	23:
		bRunSteamBypass													:= P_U01.SP_steam_bypass_immediately_after_warm_up;
		IF bAdsorptionActive AND NOT bRunSteamBypass THEN 																	// 14
			i2Step														:= 30;
		ELSIF bAdsorptionActive AND bRunSteamBypass AND NOT P_U01.SP_adsorb_during_steam_bypass THEN
			i2Step														:= 40;												// 15
		ELSE
			i2Step														:= 90;												// 13 & 16
		END_IF
	
		
//**** Adsorption 1		
	30:
		IF tonAdsorptionTimer.Q THEN																						// 14.a
			bAdsorptionTimer											:= FALSE;
			gsCycleStage												:= 'warm_up.boiler_heating.turn_off_fans';			// 14.b
			P_M01.rs1.fan_setpoint										:= 0;												// 14.c
			rTime														:= _FAN_RS_DELAY_TIME;
			i2Step														:= i2Step + 1;
		END_IF

	31:
		bTimer															:= TRUE;
		IF tonTimer.Q THEN
			bTimer														:= FALSE;
			gsCycleStage												:= 'warm_up.boiler_heating.closing_doors';			// 14.d
			P_M01.rs1.close_doors										:= TRUE;											// 14.e
			rTime														:= P_M01.SP_doorsopenclose_timedelay * _MINUTES;										// 14.e.i
			i2Step														:= i2Step + 1;
		END_IF		

	32:
		bTimer															:= TRUE;
		bPass1															:= (P_M01.bRS01 AND P_M01.rs1.inlet_doors_closed AND P_M01.rs1.outlet_doors_closed) OR NOT P_M01.bRS01;	// 14.e.ii
		IF bPass1 THEN
			bTimer														:= FALSE;
			i2Step														:= i2Step + 1;
		ELSIF tonTimer.Q THEN																								// 14.e.i
			bTimer														:= FALSE;
			bRunSteamBypass												:= FALSE;
			sRS															:= _RS01;
			P_Alarms.M_Add_Alarm(F_Concat3(_U01, sRS, gsCycleStage), gsReactorDoorClosingError, gsSystemCannotRun);
			i2Step														:= i2Step + 1;
		END_IF
		
	33:
		//P_M01_RS01.co2_sensors_on										:= FALSE;											// 14.f
		bAdsorptionActive												:= FALSE;											// 14.g
		i2Step															:= 90;

	
//**** Adsorption 2	
	40:
		IF tonAdsorptionTimer.Q THEN																						// 15.a
			bAdsorptionTimer											:= FALSE;
			P_M01.rs1.fan_setpoint										:= 0;												// 15.b
			rTime														:= _FAN_RS_DELAY_TIME;
			i2Step														:= i2Step + 1;
		END_IF

	41:
		bTimer															:= TRUE;
		IF tonTimer.Q THEN
			bTimer														:= FALSE;											// 15.c
			//P_M01_RS01.co2_sensors_on									:= FALSE;
			bAdsorptionActive											:= FALSE;											// 15.d
			i2Step														:= i2Step + 1;
		END_IF
		
	42:
		P_M01.rs1.close_doors											:= TRUE;											// 15.g
		rTime															:= P_M01.SP_doorsopenclose_timedelay * _MINUTES;										// 15.g.i
		i2Step															:= i2Step + 1;

	43:
		bTimer															:= TRUE;
		bPass1															:= (P_M01.bRS01 AND P_M01.rs1.inlet_doors_closed AND P_M01.rs1.outlet_doors_closed) OR NOT P_M01.bRS01;		// 15.g.ii
		IF bPass1 THEN
			bTimer														:= FALSE;
			i2Step														:= 90;
		ELSIF tonTimer.Q THEN
			bTimer														:= FALSE;
			bRunSteamBypass												:= FALSE;
			sRS															:= _RS01;
			P_Alarms.M_Add_Alarm(F_Concat3(_U01, sRS, gsCycleStage), gsReactorDoorOpeningError, gsSystemCannotRun);
			i2Step														:= 90;
		END_IF


//**** Process error		
	80:
		P_Alarms.M_Add_Alarm(CONCAT(_U01, gsCycleStage), sError, gsProcessCannotRun);
		gsCycleStage													:= 'warm_up.error';
		i2Step															:= i2Step + 1;

//**** Stop process		
	81:
		P_U01.vacuum_pres_control_valve									:= _CLOSED;
		//P_M01_RS01.co2_sensors_on										:= FALSE;
		P_M01.rs1.fan_setpoint											:= 0;
		rTime															:= _FAN_RS_DELAY_TIME;
		i2Step															:= i2Step + 1;

	82:
		bTimer															:= TRUE;
		IF tonTimer.Q THEN
			bTimer														:= FALSE;
			P_U01.boiler_package											:= FALSE;
			P_M01.rs1.close_doors										:= P_M01.bRS01;
			rTime														:= P_M01.SP_doorsopenclose_timedelay * _MINUTES;
			i2Step														:= 90;
		END_IF
		
//**** Close process
	90:
		gsCycleStage													:= SEL(bComplete, 'warm_up.failed', 'warm_up.complete');
		bAdsorptionTimer												:= FALSE;
		P_U01.drainage_on													:= FALSE;
		rTime															:= _PROCESS_COMPLETE_TIME;
		i2Step															:= i2Step + 1;
		
	91:
		bTimer															:= TRUE;
		IF tonTimer.Q THEN
			bTimer														:= FALSE;
			gsCycleStage												:= '';
			i2Step														:= 0;
		END_IF
				

END_CASE

IF i2Step > 0 AND i2Step < 80 AND P_U01.shutdown_process THEN
	gsCycleStage														:= 'warm_up.stopping';
	i2Step																:= 81;
END_IF
END_ACTION

ACTION A03_Steam_Bypass:
// Theseus - P_U01.A03_Steam_Bypass
// Rev 1.0 - October 7, 2024

CASE i3Step OF

	0:	;

	1:	
		bComplete														:= FALSE;
		IF P_U01.warmup_complete THEN
			IF NOT P_U01.steam_bypass_complete THEN
				gsCycleStage											:= 'steam_bypass.initialize';						// 4
				sError													:= '';
				IF P_U01.product_vacuum_pres_error THEN
					sError												:= gsProductVacuumPresSensorError;
				END_IF
				i3Step													:= SEL(sError = '', 80, i3Step + 1);
			ELSE
				bComplete												:= TRUE;
				i3Step													:= 90;
			END_IF
		ELSE
			P_U01.boiler_package										:= FALSE;
			P_Alarms.M_Add_Alarm(CONCAT(_U01, gsCycleStage), gsWarmupNotRunError, gsProcessCannotRun);
			i3Step														:= 90;
		END_IF
		
	2:	
		IF P_U01.boiler_ready THEN																							// 5.a (Handled in P_U01.A_Points)
			P_U01.bCloseXVValves										:= TRUE;											// 5.b
			rTime														:= _VALVE_TIME;
			i3Step														:= i3Step + 1;
		ELSE
			sError														:= gsBoilerError;
			sMessage													:= gsRunWarmup;
			i3Step														:= 80;
		END_IF

	3:	bTimer															:= TRUE;
		bPass1															:= P_U01.vacuum_pump_inlet_valve_closed;
		IF bPass1 THEN
			bTimer														:= FALSE;
			P_U01.vacuum_pres_control_valve								:= _OPEN;											// 5.b.iii
			rTime														:= _VALVE_TIME;
			i3Step														:= i3Step + 1;
		ELSIF tonTimer.Q THEN
			bTimer														:= FALSE;
			sError														:= SEL(bPass1, '', gsProductVacuumPumpIsoValveError);
			sError														:= SEL(bPass2, sError, gsProductVacuumOutletIsoValveError);
			i3Step														:= 80;
		END_IF
		
	4:
		bTimer															:= TRUE;
		IF P_U01.vacuum_pres_control_valve_position > _VALVE_OPEN THEN
			bTimer														:= FALSE;
			P_U01.drainage_on												:= TRUE;											// 5.c
			IF bAdsorptionActive AND P_U01.SP_adsorb_during_steam_bypass THEN													// 5.b.iv
				P_M01.rs1.open_doors									:= P_M01.bRS01;
				rTime													:= P_M01.SP_doorsopenclose_timedelay * _MINUTES;
				i3Step													:= i3Step + 1;
			ELSE
				i3Step													:= i3Step + 2;
			END_IF
		ELSIF tonTimer.Q THEN
			bTimer														:= FALSE;
			sError														:= gsProductVacuumBackfeedValveError;
			i3Step														:= 80;
		END_IF

	5:
		bTimer															:= TRUE;
		bPass1															:= (P_M01.bRS01 AND P_M01.rs1.inlet_doors_open AND P_M01.rs1.outlet_doors_open) OR NOT P_M01.bRS01;	// 5.b.iv
		IF bPass1 THEN
			bTimer														:= FALSE;
			IF NOT bAdsorptionActive AND P_U01.SP_adsorb_during_steam_bypass THEN												// 6
				iAxStep													:= 1;												// 6.b
				i3Step													:= i3Step + 1;
			ELSE
				i3Step													:= 20;
			END_IF
		ELSIF tonTimer.Q THEN
			bTimer														:= FALSE;
			bAdsorptionActive											:= FALSE;
			sRS															:= _RS01;
			P_Alarms.M_Add_Alarm(F_Concat3(_U01, sRS, gsCycleStage), gsReactorDoorOpeningError, gsSteamBypassWillContinueWOAdsorption);
			i3Step														:= 20;
		END_IF

	6:
		Ax_Process_Pre_Check();																								// 6.b																			
		IF bPreCheckDone THEN
			IF sError = '' THEN																								// 6.b.i
				P_M01.rs1.repres_valves									:= P_M01.bRS01;										// 6.c
				rTime													:= _VALVE_TIME;
				i3Step													:= i3Step + 1;
			ELSE
				P_Alarms.M_Add_Alarm(CONCAT(_U01, gsCycleStage), sError, gsSteamBypassWillContinueWOAdsorption);			// 6.b.ii
				bAdsorptionActive										:= FALSE;
				i3Step													:= 20;
			END_IF
		END_IF

	7:
		bTimer															:= TRUE;
		bPass1															:= (P_M01.bRS01 AND P_M01.rs1.repres_valves_clear) OR NOT P_M01.bRS01;
		IF bPass1 AND bPass2 AND bPass3 THEN
			bTimer														:= FALSE;
			i3Step														:= i3Step + 1;
		ELSIF tonTimer.Q THEN
			bTimer														:= FALSE;
			i3Step														:= i3Step + 1;
			//bAdsorptionActive											:= FALSE;
			//P_M01_RS01.close_repres_valves								:= P_M01.bRS01;
			//i3Step													:= 20; 
		END_IF
		
	8:
		P_M01.rs1.open_doors											:= P_M01.bRS01;
		gsCycleStage													:= 'steam_bypass.initialize.open_doors';			// 6.d.ii
		rTime															:= P_M01.SP_doorsopenclose_timedelay * _MINUTES;										// 6.d.i
		i3Step															:= i3Step + 1;

	9:
		bTimer															:= TRUE; 
		bPass1															:= (P_M01.bRS01 AND P_M01.rs1.inlet_doors_open AND P_M01.rs1.outlet_doors_open) OR NOT P_M01.bRS01;	// 6.d.ii
		IF bPass1 AND bPass2 AND bPass3 THEN
			bTimer														:= FALSE;
			i3Step														:= i3Step + 1;
		ELSIF tonTimer.Q THEN
			bTimer														:= FALSE;
			sRS															:= _RS01;
			P_Alarms.M_Add_Alarm(F_Concat3(_U01, sRS, gsCycleStage), gsReactorDoorOpeningError, gsSteamBypassWillContinueWOAdsorption);
			bAdsorptionActive											:= FALSE;
			i3Step														:= 20;
		END_IF

	10:
		P_M01.rs1.fan_setpoint											:= SEL(P_M01.bRS01, 0, P_M01.SP_reactor_set_1_vfd_percent);	// 6.e
		gsCycleStage													:= 'steam_bypass.initialize.turn_on_fans';			// 6.e.i
		rTime															:= _FAN_RS_DELAY_TIME;
		i3Step															:= i3Step + 1;

	11:
		bTimer															:= TRUE;
		IF tonTimer.Q THEN
			bTimer														:= FALSE;
			i3Step														:= i3Step + 1;
		END_IF

	12:
		//P_M01_RS01.co2_sensors_on										:= P_M01.bRS01;										// 6.f
		gsCycleStage													:= 'steam_bypass.initialize.adsorption';			// 6.f.i
		bAdsorptionTimer												:= TRUE;											// 6.a
		bAdsorptionActive												:= TRUE;											// 6.g
		i3Step															:= 20;


//**** Complete Steam Bypass		
	20:
		rSP																:= P_U01.SP_steam_bypass_vacuum_pressure;				// 8
		bPass1															:= P_U01.product_vacuum_pres < rSP;
		bPass2															:= P_U01.product_vacuum_pres < rSP;
		i3Step															:= SEL(bPass1 AND bPass2, i3Step + 1, 30);
	
	21:
		P_U01.vacuum_pump_inlet_valve										:= TRUE;											// 9.a
		rTime															:= _VALVE_TIME;
		i3Step															:= i3Step + 1;
		
	22:
		bTimer															:= TRUE;
		bPass1															:= P_U01.vacuum_pump_inlet_valve_open;
		IF bPass1 AND bPass2 THEN
			bTimer														:= FALSE;
			//P_U01.fan											:= TRUE;											// 9.a
			P_U01.vacuum_pres_control_valve								:= _CLOSED;
			i3Step														:= i3Step + 1;
		ELSIF tonTimer.Q THEN
			bTimer														:= FALSE;
			sError														:= SEL(bPass1, '', gsProductVacuumPumpIsoValveError);
			sError														:= SEL(bPass2, sError, gsProductVacuumOutletIsoValveError);
			i3Step														:= 80;
		END_IF
		
	23:	
		gsCycleStage													:= SEL(bAdsorptionActive, 'steam_bypass.evacuate_lines', 'steam_bypass.evacuate_lines.adsorption');		// 9.b.i
		rTime															:= P_M01.SP_evacuation_duration * _MINUTES;
		i3Step															:= i3Step + 1;
		
	24:
		bTimer															:= TRUE;											// 9.d
		rSP																:= P_U01.SP_steam_bypass_vacuum_pressure;
		bPass1															:= P_U01.product_vacuum_pres < rSP;
		bPass2															:= P_U01.product_vacuum_pres < rSP;
		IF bPass1 AND bPass2 THEN
			bTimer														:= FALSE;
			i3Step														:= i3Step + 1;
		ELSIF tonTimer.Q THEN
			bTimer														:= FALSE;
			sError														:= gsUnableToEvacuateLinesError;
			i3Step														:= 80;
		END_IF
	
	25:	
		P_U01.vacuum_pump_inlet_valve										:= FALSE;											// 9.e
		P_U01.vacuum_pres_control_valve									:= _OPEN;
		//P_U01.fan											:= FALSE;
		i3Step															:= 30;

		
//**** Steam Bypass		
	30:
		//P_U01.steam_bypass_valve											:= TRUE;											// 10
		gsCycleStage													:= SEL(bAdsorptionActive, 'steam_bypass.steam_bypass.adsorption', 'steam_bypass.steam_bypass');		// 10.a
		rSP																:= P_U01.SP_steam_bypass_duration * _MINUTES;				
		rTime															:= rSP;
		i3Step															:= i3Step + 1;				

	31:
		i3Step															:= i3Step + 1;
		
	32:
		P_U01.vacuum_pump_bypass_valve									:= TRUE;											// 12
		//P_U01.fan												:= TRUE;
		i3Step															:= i3Step + 1;
		
	33:
		IF TIME_TO_REAL(tonTimer.ET) >= (rSP * 0.3) THEN																	// 13
			i3Step														:= i3Step + 1;
		END_IF 
	
	34:
		i3Step															:= i3Step + 1;										// 13.a
	
	35:
		IF tonTimer.Q THEN //OR P_U01.product_line_temp > P_U01.SP_steam_bypass_temperature THEN										// 14
			bTimer														:= FALSE;
			//P_U01.steam_bypass_valve										:= FALSE;											// 15
			gsCycleStage												:= SEL(bAdsorptionActive, 'steam_bypass.wrap_up', 'steam_bypass.wrap_up.adsorption');	// 15.a
			P_U01.vacuum_pump_bypass_valve								:= FALSE;
			//P_U01.fan											:= FALSE;
			IF bAdsorptionActive THEN
				i3Step													:= 40;
			ELSE
				P_U01.steam_bypass_complete								:= TRUE;
				i3Step													:= 90;
			END_IF
		END_IF
		
		
//**** Complete Adsorption		
	40:
		IF tonAdsorptionTimer.Q THEN																						// 17.a.i
			bAdsorptionTimer											:= FALSE;
			P_M01.rs1.fan_setpoint										:= 0;												// 17.a.ii
			gsCycleStage												:= 'steam_bypass.wrap_up.turn_off_fans';			// 17.a.ii.1
			rTime														:= _FAN_RS_DELAY_TIME;
			i3Step														:= i3Step + 1;
		END_IF

	41:
		bTimer															:= TRUE;
		IF tonTimer.Q THEN
			bTimer														:= FALSE;
			P_M01.rs1.close_doors										:= TRUE;											// 17.a.iii
			gsCycleStage												:= 'steam_bypass.wrap_up.close_doors';				// 17.a.iii.1
			rTime														:= P_M01.SP_doorsopenclose_timedelay * _MINUTES;										// 17.a.iii.2
			i3Step														:= i3Step + 1;
		END_IF		

	42:
		bTimer															:= TRUE;
		bPass1															:= (P_M01.bRS01 AND P_M01.rs1.inlet_doors_closed AND P_M01.rs1.outlet_doors_closed) OR NOT P_M01.bRS01;		// 17.a.iii.3
		IF bPass1 AND bPass2 AND bPass3 THEN
			bTimer														:= FALSE;
			i3Step														:= i3Step + 1;
		ELSIF tonTimer.Q THEN
			bTimer														:= FALSE;
			sRS															:= _RS01;
			P_Alarms.M_Add_Alarm(F_Concat3(_U01, sRS, gsCycleStage), gsReactorDoorClosingError, gsSystemCannotRun);
			i3Step														:= i3Step + 1;
		END_IF
		
	43:
		//P_M01_RS01.co2_sensors_on										:= FALSE;											// 17.a.iv
		bAdsorptionActive												:= FALSE;											// 17.a.v
		i3Step															:= 90;

	
//**** Process error		
	80:
		gsCycleStage													:= 'steam_bypass.error';
		sMessage														:= SEL(sMessage = gsRunWarmup, gsProcessCannotRun, sMessage);
		P_Alarms.M_Add_Alarm(CONCAT(_U01, gsCycleStage), sError, sMessage);
		i3Step															:= i3Step + 1;

//**** Stop process
	81:
		//P_M01_RS01.co2_sensors_on										:= FALSE;
		P_M01.rs1.fan_setpoint											:= 0;
		rTime															:= _FAN_RS_DELAY_TIME;
		i3Step															:= i3Step + 1;

	82:
		bTimer															:= TRUE;
		IF tonTimer.Q THEN
			bTimer														:= FALSE;
			i3Step														:= i3Step + 1;
		END_IF

	83:
		//P_U01.fan												:= FALSE;
		P_U01.vacuum_pump_bypass_valve									:= FALSE;
		P_U01.vacuum_pres_control_valve									:= _CLOSED;
		P_U01.vacuum_pump_inlet_valve									:= FALSE;
		rTime															:= _VALVE_TIME;
		i3Step															:= i3Step + 1;
		
	84:
		bTimer															:= TRUE;
		IF tonTimer.Q THEN
			bTimer														:= FALSE;
			i3Step														:= 90;
		END_IF
		
//**** Close process
	90:
		gsCycleStage													:= SEL(bComplete, 'steam_bypass.failed', 'steam_bypass.complete');
		bAdsorptionTimer												:= FALSE;
		P_U01.drainage_on												:= FALSE;
		rTime															:= _PROCESS_COMPLETE_TIME;
		i3Step															:= i3Step + 1;
		
	91:
		bTimer															:= TRUE;
		IF tonTimer.Q THEN
			bTimer														:= FALSE;
			gsCycleStage												:= '';
			i3Step														:= 0;
		END_IF
				
END_CASE

IF i3Step > 0 AND i3Step < 80 AND P_U01.shutdown_process THEN
	gsCycleStage														:= 'steam_bypass.stopping';
	i3Step																:= 81;
END_IF
END_ACTION

ACTION A08_Shutdown:
// Theseus - P_U01.A08_Shutdown
// Rev 1.0 - October 7, 2024

CASE i8Step OF

	0:	;

	1:	
		bComplete														:= FALSE;
		gsCycleStage													:= 'shutdown.initialize';							// 1.a
		P_U01.boiler_package												:= FALSE;											// 3
		i8Step															:= i8Step + 1;

	2:
		P_M01.rs1.fan_setpoint											:= 0;
		rTime															:= _PAUSE_TIME;
		i8Step															:= i8Step + 1;
		
	3:
		bTimer															:= TRUE;
		IF tonTimer.Q THEN
			bTimer														:= FALSE;						
			P_M01.rs1.close_doors										:= P_M01.bRS01;										// 4
			gsCycleStage												:= 'shutdown.close_doors';							// 4.a
			rTime														:= P_M01.SP_doorsopenclose_timedelay * _MINUTES;
			i8Step														:= i8Step + 1;
		END_IF

	4:
		bTimer															:= TRUE; 
		bPass1															:= (P_M01.bRS01 AND P_M01.rs1.inlet_doors_closed AND P_M01.rs1.outlet_doors_closed) OR NOT P_M01.bRS01;
		IF bPass1 OR tonTimer.Q THEN
			IF tonTimer.Q THEN 
				sRS														:= _RS01;
				P_Alarms.M_Add_Alarm(F_Concat3(_U01, gsCycleStage, sRS), gsReactorDoorClosingError, gsSystemCannotRun);
			END_IF
			bTimer														:= FALSE;
			i8Step														:= i8Step + 1;
		END_IF

	5:
		P_M01.rs1.close_valves											:= P_M01.bRS01;										// 5		
		gsCycleStage													:= 'shutdown.wrap_up';								// 5.a
		rTime															:= _VALVE_TIME;
		i8Step															:= i8Step + 1;
		
	6:
		bTimer															:= TRUE;
		IF tonTimer.Q THEN
			bTimer														:= FALSE;
			//P_M01_RS01.co2_sensors_on									:= NOT P_M01.bRS01;
			P_M01.rs1.repres_valves										:= NOT P_M01.bRS01;
			i8Step														:= i8Step + 1;
		END_IF
		
	7:
		P_U01.bCloseXVValves											:= TRUE;
		P_U01.vacuum_pres_control_valve									:= 0;
		rTime															:= _PAUSE_TIME;
		i8Step															:= i8Step + 1;

	8:
		bTimer															:= TRUE;
		bPass1															:= NOT P_M01.rs1.reactor_drain_vessel_lsl;			// 6
		bPass2															:= NOT product_condensate_drum_lsh;
		gsCycleStage													:= 'shutdown.drain';								// 6.a
		IF bPass1 AND bPass2 THEN
			bTimer														:= FALSE;
 		ELSIF tonTimer.Q THEN
			sError														:= SEL(NOT bPass1, '', F_concat3(_RS01, ' ', gsCondensateLslError));
			sError														:= SEL(NOT bPass2, sError, gsProductCondensateDrumLshError);
			P_Alarms.M_Add_Alarm(_U01, sError, gsCheckOperation);
		END_IF
		i8Step															:= 90;
		
//**** Close process
	90:
		gsCycleStage													:= 'shutdown.complete';								// 7
		rTime															:= _PROCESS_COMPLETE_TIME;
		i8Step															:= i8Step + 1;
		
	91:
		bTimer															:= TRUE;
		IF tonTimer.Q THEN
			bTimer														:= FALSE;
			gsCycleStage												:= '';
			i8Step														:= 0;
		END_IF
				
END_CASE

IF i8Step > 0 AND i8Step < 80 AND P_U01.shutdown_process THEN
	gsCycleStage														:= 'shutdown.stopping';
	i8Step																:= 81;
END_IF
END_ACTION

ACTION A09_Pressure_Drop_Test:
// Theseus - P_U01.A09_Pressure_Drop_Test
// Rev 1.0 - October 8, 2024

CASE i9Step OF

	0:	;

	1:	
		bComplete														:= FALSE;
		gsCycleStage													:= 'pressure_drop_test.initialize';					// 3
		i9Step															:= i9Step + 1;

	2:	
		Ax_Process_Pre_Check();																								// 3.a																			
		IF bPreCheckDone THEN
			IF sError = '' THEN																								// 3.a.i
				P_U01.drainage_on											:= TRUE;											// 3.c
				i9Step													:= i9Step + 1;
			ELSE
				sRS														:= '';
				sMessage												:= gsPressureDropTestCannotRun;						// 3.a.ii
				i9Step													:= 80;
			END_IF
		END_IF

	3:
		P_M01.rs1.repres_valves											:= P_M01.bRS01;										// 4
		rTime															:= _VALVE_TIME;
		i9Step															:= i9Step + 1;

	4:
		bTimer															:= TRUE;
		bPass1															:= (P_M01.bRS01 AND P_M01.rs1.repres_valves_clear) OR NOT P_M01.bRS01;
		IF bPass1 OR tonTimer.Q THEN
			bTimer														:= FALSE;
			i9Step														:= i9Step + 1;
		END_IF
		
	5:
		P_M01.rs1.open_doors											:= P_M01.bRS01;										// 5
		gsCycleStage													:= 'pressure_drop_test.open_doors';					// 5.a
		rTime															:= P_M01.SP_doorsopenclose_timedelay * _MINUTES;		// 5.b
		i9Step															:= i9Step + 1;

	6:
		bTimer															:= TRUE; 
		bPass1															:= (P_M01.bRS01 AND P_M01.rs1.inlet_doors_open AND P_M01.rs1.outlet_doors_open) OR NOT P_M01.bRS01;	// 5.c
		IF bPass1 THEN
			bTimer														:= FALSE;
			iVfd_Speed													:= P_U01.SP_reactor_vfd_percent_step_size;			// 6
			bVfd_Speed_Up												:= TRUE;
			gsCycleStage												:= 'pressure_drop_test.pressure_drop_test';			// 6.a
			rTime														:= P_U01.SP_reactor_vfd_percent_step_duration * _MINUTES;	// 7
			i9Step														:= i9Step + 1;
		ELSIF tonTimer.Q THEN
			bTimer														:= FALSE;
			sRS															:= _RS01;
			sError														:= gsReactorDoorOpeningError;
			sMessage													:= gsPressureDropTestCannotRun;
			i9Step														:= 80;
		END_IF

	7:
		P_M01.rs1.fan_setpoint											:= SEL(P_M01.bRS01, 0, iVfd_Speed);
		i9Step															:= SEL(iVfd_Speed = 0, i9Step + 1, i9Step + 2);		//11

	8:
		bTimer															:= TRUE;
		IF tonTimer.Q THEN																									// 8
			bTimer														:= FALSE;
			IF bVfd_Speed_Up THEN
				IF iVfd_Speed + P_U01.SP_reactor_vfd_percent_step_size <= P_U01.SP_reactor_vfd_percent_maximum THEN
					iVfd_Speed											:= iVfd_Speed + P_U01.SP_reactor_vfd_percent_step_size;	// 9
				ELSE
					bVfd_Speed_Up										:= FALSE;
					iVfd_Speed											:= iVfd_Speed - P_U01.SP_reactor_vfd_percent_step_size;
				END_IF
			ELSE
				IF iVfd_Speed - P_U01.SP_reactor_vfd_percent_step_size >= 0 THEN
					iVfd_Speed											:= iVfd_Speed - P_U01.SP_reactor_vfd_percent_step_size;	// 10
				ELSE
					iVfd_Speed											:= 0;
				END_IF
			END_IF
			i9Step														:= i9Step - 1;
		END_IF

	9:
		bComplete														:= TRUE;
		gsCycleStage													:= 'pressure_drop_test.close_doors';				// 11.a
		P_M01.rs1.close_doors											:= P_M01.bRS01;										// 12
		rTime															:= P_M01.SP_doorsopenclose_timedelay * _MINUTES;										// 12.a
		i9Step															:= i9Step + 1;

	10:
		bTimer															:= TRUE;
		bPass1															:= (P_M01.bRS01 AND P_M01.rs1.inlet_doors_closed and P_M01.rs1.outlet_doors_closed) OR NOT P_M01.bRS01;	// 12.b
		IF bPass1 THEN
			bTimer														:= FALSE;
			i9Step														:= i9Step + 1;
		ELSIF tonTimer.Q THEN
			bTimer														:= FALSE;
			sRS															:= _RS01;
			P_Alarms.M_Add_Alarm(F_Concat3(_U01, gsCycleStage, sRS), gsReactorDoorClosingError, gsUnableToCloseDoors);
			i9Step														:= 90;
		END_IF
		

//**** Process error		
	80:
		gsCycleStage													:= 'pressure_drop_test.error';
		P_Alarms.M_Add_Alarm(F_Concat3(_U01, sRS, gsCycleStage), sError, sMessage);
		i9Step															:= i9Step + 1;

//**** Stop process		
	81:
		P_M01.rs1.fan_setpoint											:= 0;
		i9Step															:= 90;
		
//**** Close process
	90:
		gsCycleStage													:= SEL(bComplete, 'pressure_drop_test.failed', 'pressure_drop_test.complete');	// 13
		P_U01.drainage_on													:= FALSE;
		rTime															:= _PROCESS_COMPLETE_TIME;
		i9Step															:= i9Step + 1;
		
	91:
		bTimer															:= TRUE;
		IF tonTimer.Q THEN
			bTimer														:= FALSE;
			gsCycleStage												:= '';
			i9Step														:= 0;
		END_IF
				
END_CASE

IF i9Step > 0 AND i9Step < 80 AND P_U01.shutdown_process THEN
	gsCycleStage														:= 'pressure_drop_test.stopping';
	i9Step																:= 81;
END_IF
END_ACTION

ACTION Ax_Process_Pre_Check:
// Theseus - P_U01.Ax_Process_Pre_Check
// Rev 1.0 - October 7, 2024

CASE iAxStep OF

	0:	;

	1:	
		sError															:= '';
		bPreCheckDone													:= FALSE;
		P_M01.rs1.close_valves											:= P_M01.bRS01;
		P_M01.rs1.retract_clamps										:= P_M01.bRS01;
		rTime															:= _VALVE_TIME;
		iAxStep															:= iAxStep + 1;
	
	2:	
		bTimer															:= TRUE;
		bPass1															:= (P_M01.bRS01 AND P_M01.rs1.rs_valves_clear) OR NOT P_M01.bRS01;
		IF bPass1 THEN
			bTimer														:= FALSE;
			iAxStep														:= iAxStep + 1;
		ELSIF tonTimer.Q THEN
			sError														:= 'Valve Error';
			iAxStep														:= 99;
		END_IF

	3:
		IF P_M01.rs1.adsorption_high_temp_count <= _HIGH_CART_READINGS_MAX THEN
			iAxStep														:= iAxStep + 1;
		ELSE
			sError														:= gsHighTempCountError;
			iAxStep														:= 99;
		END_IF

	4:
		bPass1															:= (P_M01.bRS01 AND P_M01.rs1.inlet_clamps_retracted) OR NOT P_M01.bRS01; 
		IF bPass1 AND bPass2 AND bPass3 THEN
			iAxStep														:= iAxStep + 1;
		ELSE
			sError														:= gsClampRetractError;
			iAxStep														:= 99;
		END_IF
		
	5:
		iAxStep															:= iAxStep + 1;
		
	6:
		///@@@bPass1															:= (P_M01.bRS01 AND P_M01.rs1.average_pressure_within_ambient) OR NOT P_M01.bRS01;
		IF NOT bPass1 OR NOT bPass2 OR NOT bPass3 THEN
			sError														:=  gsAmbientPressureError;
		END_IF
		iAxStep															:= 99;
		
	99:
		bTimer															:= FALSE;
		bPreCheckDone													:= TRUE;
		iAxStep															:= 0;
				
END_CASE
END_ACTION

END_PROGRAM

(* stored: Version 1.1.0.1, ProductVersion 3.1.4024.12
   POU P_U01: Id {dcf8449b-3592-47e4-a482-48f13716f004}, SpecialFunc None
   Action A_IO_Points: Id {d2567efd-8816-46e7-a69d-41abdef6a01f}
   Action A_MovingAverage: Id {8485b6cb-e244-43cb-929b-696de39510b1}
   Action A_PIDs: Id {bdad273d-c5b6-4cdc-9e45-b9c5a8ce2ca9}
   Action A02_WarmUp: Id {3e02c609-752d-4440-9a0e-94c91ce7baf7}
   Action A03_Steam_Bypass: Id {73856173-8e49-4891-b8be-3c57dfbf2633}
   Action A08_Shutdown: Id {dceaad34-9fba-494d-9502-9d4c836ba12b}
   Action A09_Pressure_Drop_Test: Id {b8bf7e66-dcdb-4668-8218-16ff48a3e793}
   Action Ax_Process_Pre_Check: Id {d59aaf0d-9d27-45c8-bc13-c9bb5b8aaff8} *)
